Staubli VAL3: test.pjx

--- test.pjx ---
Parameters version=s7.10 stackSize=5000 millimeterUnit=true
Program file=inicializar.pgx
Program file=mcp.pgx
Program file=Pick.pgx
Program file=Piramide.pgx
Program file=place.pgx
Program file=start.pgx
Program file=stop.pgx
Data file=test.dtx

--- test.dtx ---
mdesc mNomSpeed
mdesc mVelApprox = {accel=25, vel=50, decel=25, blend=off}
num nHPieza = 12
num nLMesa = 400
num nLPieza = 69
num nWMesa = 300
num nWPieza = 23
tool tVentosa = {z=22, fatherId=flange[0], ioLink=valve1, ioOpen=0.5, ioClose=0.5}
pointRx pCentro = {fatherId=world[0]}
pointRx pPieza = {fatherId=world[0]}
num nPlantas
num nNivel
num nFila
pointRx pObjetivo = {fatherId=world[0]}
num nX
num nY
num nZ
bool bStartPiramide
bool bTermina
jointRx jHome
bool bFin
num nTecla
string sMensaje
bool bPiezaPreparada
num nCont
num nPlantasListas

--- start.pgx ---
program start()
begin
  // Se pone en marcha la aplicacion

  // Se inicializar la aplicacion
  call inicializar()

  taskCreate "Pirámide",100,Piramide()
  taskCreate "mcp",100,mcp()
end

--- inicializar.pgx ---
program inicializar()
begin

  // Booleanos
  bPiezaPreparada=false
  bFin=false
  bTermina=false
  bStartPiramide=false

  // Variables Pieza
  // Longitud
  nLPieza=71
  // Ancho
  nWPieza=25
  // Altura
  nHPieza=12

  // Variables mesa de trabajo
  nLMesa=400
  nWMesa=300

  // Variables y contadores usados
  nPlantas=0 // Plantas introducidas por usuario
  nNivel=0 // Planta actual
  nFila=0 // Fila actual
  nCont=0 // Contador para variación de fila
  nX=0 // Variación en x (fila)
  nY=0 // Variación en y (pieza de la fila)
  nZ=2 // Variación en z (nivel). Valor = margen de error

  sMensaje="" //Mensaje a mostrar en pantalla

  // Sistema de referencia
  pCentro=appro(pPieza,{(nWMesa/2-nWPieza/2),-(nLMesa/2-nLPieza/2),0,0,0,0})

end

--- mcp.pgx ---
program mcp()
begin

  title("Pirámide")

  userPage()

  while !bFin
    // Se borra la pantalla
    cls()

    // Se muestra informacion en la pantalla
    gotoxy(2,3)
    put("Total  = "+toString("4",nPlantas))
    gotoxy(2,4)
    put("Actual = "+toString("4",nNivel))
    gotoxy(7,7)
    put(sMensaje)

    // Se muestran las etiquetas de las teclas de funcion
    gotoxy(0,13)
    put("Pir.")
    gotoxy(10,13)
    put("Edit")
    gotoxy(35,13)
    put("Fin")

    // Se procesa la tecla pulsada
    nTecla=getKey()
    switch nTecla
      // Enter - Orden de continuar
      case 270
        bPiezaPreparada=true
      break
      // F1 - Orden de construir piramide
      case 271
        bStartPiramide=true
      break
      // F3 - Orden de editar el numero de plantas a construir
      case 273
        //Obtener n
        gotoxy(1,1)
        put("Introduzca nº plantas")
        gotoxy(23,1)
        get(nPlantas)
      break
      // F8 - Orden de salir de la aplicacion
      case 278
        bTermina=true
      break
    endSwitch
    // Se da paso a la siguiente tarea y se estabiliza la pantalla
    delay(0.1)
  endWhile
  bFin=false
  // Se muestra un mensaje de despedida
  cls()
  gotoxy(12,7)
  put("Programa terminado")

end

--- Pick.pgx ---
program pick(point pPosition, tool tTool, mdesc mApproach, mdesc mTarget)
  local point pOffset
begin

  // Función para coger la pieza desde el punto donde se alimenta
  pOffset=appro(pPosition,{0,0,-50,0,0,0})
  movej(pOffset,tTool,mApproach) // Se aproxima al destino
  movel(pPosition,tTool,mTarget)
  close(tTool)
  movel(pOffset,tTool,mTarget)

end

--- Piramide.pgx ---
program Piramide()
  local num j
  local num k
  local num i
  local num l
begin
  //Mueve el brazo para crear una pirámide en 3D.

  // Se desplaza a la posicion de espera
  pEspera=appro(pPieza,{0,0,-50,0,0,0})
  movej(pEspera,tVentosa,mNomSpeed)
  waitEndMove()

  //Ciclo
  while !bTermina
    if bStartPiramide
      for i = 0 to nPlantas - 1 // Bucle de plantas
        for j = 0 to nPlantas - nNivel - 1 // Bucle de filas
          for k = 0 to nPlantas - nNivel - nFila - 1 // Bucle de piezas para fila central y superiores
            // Se espera la orden de pieza preparada para continuar
            sMensaje="pulse 'enter' para continuar"
            wait(bPiezaPreparada)
            bPiezaPreparada=false
            sMensaje=""

            pObjetivo = appro(pCentro,{nX,(nLPieza/2)*(nPlantas-nNivel-nFila-1)-nY,-nZ,0,0,0})
            call pick(pPieza,tVentosa,mNomSpeed,mVelApprox)
            call place(pObjetivo,tVentosa,mNomSpeed,mVelApprox)
            nY=nY+nLPieza
          endFor
          // Nueva fila, se reinician los valores de nY y aumenta nCont que calcula un nuevo valor para nX
          nY=0
          nCont=nCont+1
          //nX aumenta para hacer una fila inferior a continuación
          nX=nX+nWPieza*nCont
          //Aumenta nFila para disminuir nº de piezas por cada fila
          nFila=nFila+1
          for l = 0 to nPlantas - nNivel - nFila - 1 // Se repite el bucle de piezas para hacer también las filas inferiores
            // Se espera la orden de pieza preparada para continuar
            sMensaje="pulse 'enter' para continuar"
            wait(bPiezaPreparada)
            bPiezaPreparada=false
            sMensaje=""

            pObjetivo = appro(pCentro,{nX,(nLPieza/2)*(nPlantas-nNivel-nFila-1)-nY,-nZ,0,0,0})
            call pick(pPieza,tVentosa,mNomSpeed,mVelApprox)
            call place(pObjetivo,tVentosa,mNomSpeed,mVelApprox)
            nY=nY+nLPieza
          endFor
          // Nueva fila, se reinician los valores de nY y aumenta nCont que calcula un nuevo valor para nX
          nY=0
          nCont=nCont+1
          //nX disminuye para hacer una fila superior a continuación
          nX=nX-nWPieza*nCont
        endFor
        //Nueva planta, se reinician los valores nX, nFila y nCont y aumentan nZ y nNivel
        nX=0
        nZ=nZ+12
        nFila=0
        nCont=0
        nNivel=nNivel+1
      endFor
      bStartPiramide=false
    endIf
    delay(0) // Se le da paso a la siguiente tarea
  endWhile
  bTermina=false

  // Se vuelve a la posición de orgien
  movej(jHome,tVentosa,mNomSpeed)
  waitEndMove()

  bFin=true

end

--- place.pgx ---
program place(point pPosition, tool tTool, mdesc mApproach, mdesc mTarget)
  local point pOffset
begin

  // Función para soltar la pieza en el lugar deseado
  pOffset=appro(pPosition,{0,0,-50,0,0,0})
  movej(pOffset,tTool,mApproach) // Se aproxima al destino
  movel(pPosition,tTool,mTarget)
  open(tTool)
  movel(pOffset,tTool,mTarget)

end
